PROGRAM MAIN
VAR
	counterA:INT;
	counter2:INT;
	useless_variable:BOOL;
	useless_variable3:REAL;
END_VAR

counterA:=counterA+1;
counter2:=counter2+1;

END_PROGRAM

(* stored: Version 1.1.0.1, ProductVersion 3.1.4024.9
   POU MAIN: Id {d11ea297-e766-42ef-a2af-be53d91dcc2d}, SpecialFunc None *)
